PROGRAM Axis03_Manual
VAR
	Always_ON	:	BOOL	:=TRUE	;//상시 ON 
	Always_OFF	:	BOOL	:=FALSE	;//상시 OFF
END_VAR

// NETWORK 1

END_PROGRAM

(* stored: Version 1.1.0.1, ProductVersion 3.1.4024.15
   POU Axis03_Manual: Id {b3baa510-4996-43fa-9116-f4c7f51d64b4}, SpecialFunc None *)
